Fanuc KAREL source: kd00027.KL

-- PROVISIONAL review KL for V770-1; original PC SHA256 3a943ad53352f596d63e49e3e264b62fc33890ac063e2433768613d4afb82c99
-- Incomplete behavior may be omitted. Consult companion uncertainty JSON. Do not deploy.
PROGRAM KD00027
%NOLOCKGROUP
VAR
  I : INTEGER
  J : INTEGER
  B : BOOLEAN
  R : REAL
  S : STRING[80]
BEGIN
  -- UNRESOLVED_PC offsets 5-21; opcodes 9D,81,18,9D,12,22,9D,13,04
  -- UNRESOLVED_PC offsets 26-30; opcodes 7F
END KD00027
